// TIA Portal V19 export
FUNCTION "FC_EM_General" : Void   // FC1, FBD
TITLE = FC Algemeen
{ S7_Optimized_Access := 'TRUE' }
// stored: SetENOAutomatically false
   VAR_TEMP
      xFlashPeriod : Real;
   END_VAR
BEGIN

REGION Network 1: ------------------------------------------------------------------------ Inputs ------------------------------------------------------------------------
END_REGION

REGION Network 2: Verwerken van iStsNoodstop
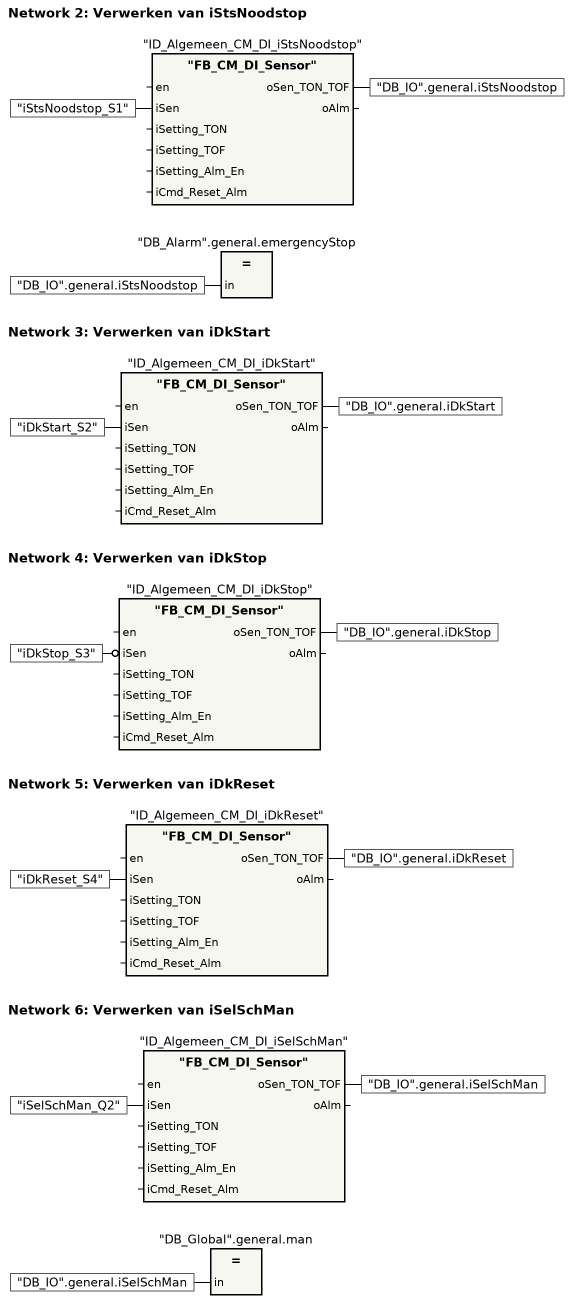
   "ID_Algemeen_CM_DI_iStsNoodstop"(iSen := "iStsNoodstop_S1", oSen_TON_TOF => "DB_IO".general.iStsNoodstop);   // "FB_CM_DI_Sensor"
   "DB_Alarm".general.emergencyStop := "DB_IO".general.iStsNoodstop;
END_REGION

REGION Network 3: Verwerken van iDkStart
   "ID_Algemeen_CM_DI_iDkStart"(iSen := "iDkStart_S2", oSen_TON_TOF => "DB_IO".general.iDkStart);   // "FB_CM_DI_Sensor"
END_REGION

REGION Network 4: Verwerken van iDkStop
   "ID_Algemeen_CM_DI_iDkStop"(iSen := NOT "iDkStop_S3", oSen_TON_TOF => "DB_IO".general.iDkStop);   // "FB_CM_DI_Sensor"
END_REGION

REGION Network 5: Verwerken van iDkReset
   "ID_Algemeen_CM_DI_iDkReset"(iSen := "iDkReset_S4", oSen_TON_TOF => "DB_IO".general.iDkReset);   // "FB_CM_DI_Sensor"
END_REGION

REGION Network 6: Verwerken van iSelSchMan
   "ID_Algemeen_CM_DI_iSelSchMan"(iSen := "iSelSchMan_Q2", oSen_TON_TOF => "DB_IO".general.iSelSchMan);   // "FB_CM_DI_Sensor"
   "DB_Global".general.man := "DB_IO".general.iSelSchMan;
END_REGION

REGION Network 7: ------------------------------------------------------------------------ Logic -------------------------------------------------------------------------
END_REGION

REGION Network 8: Start/stop logica van de installatie
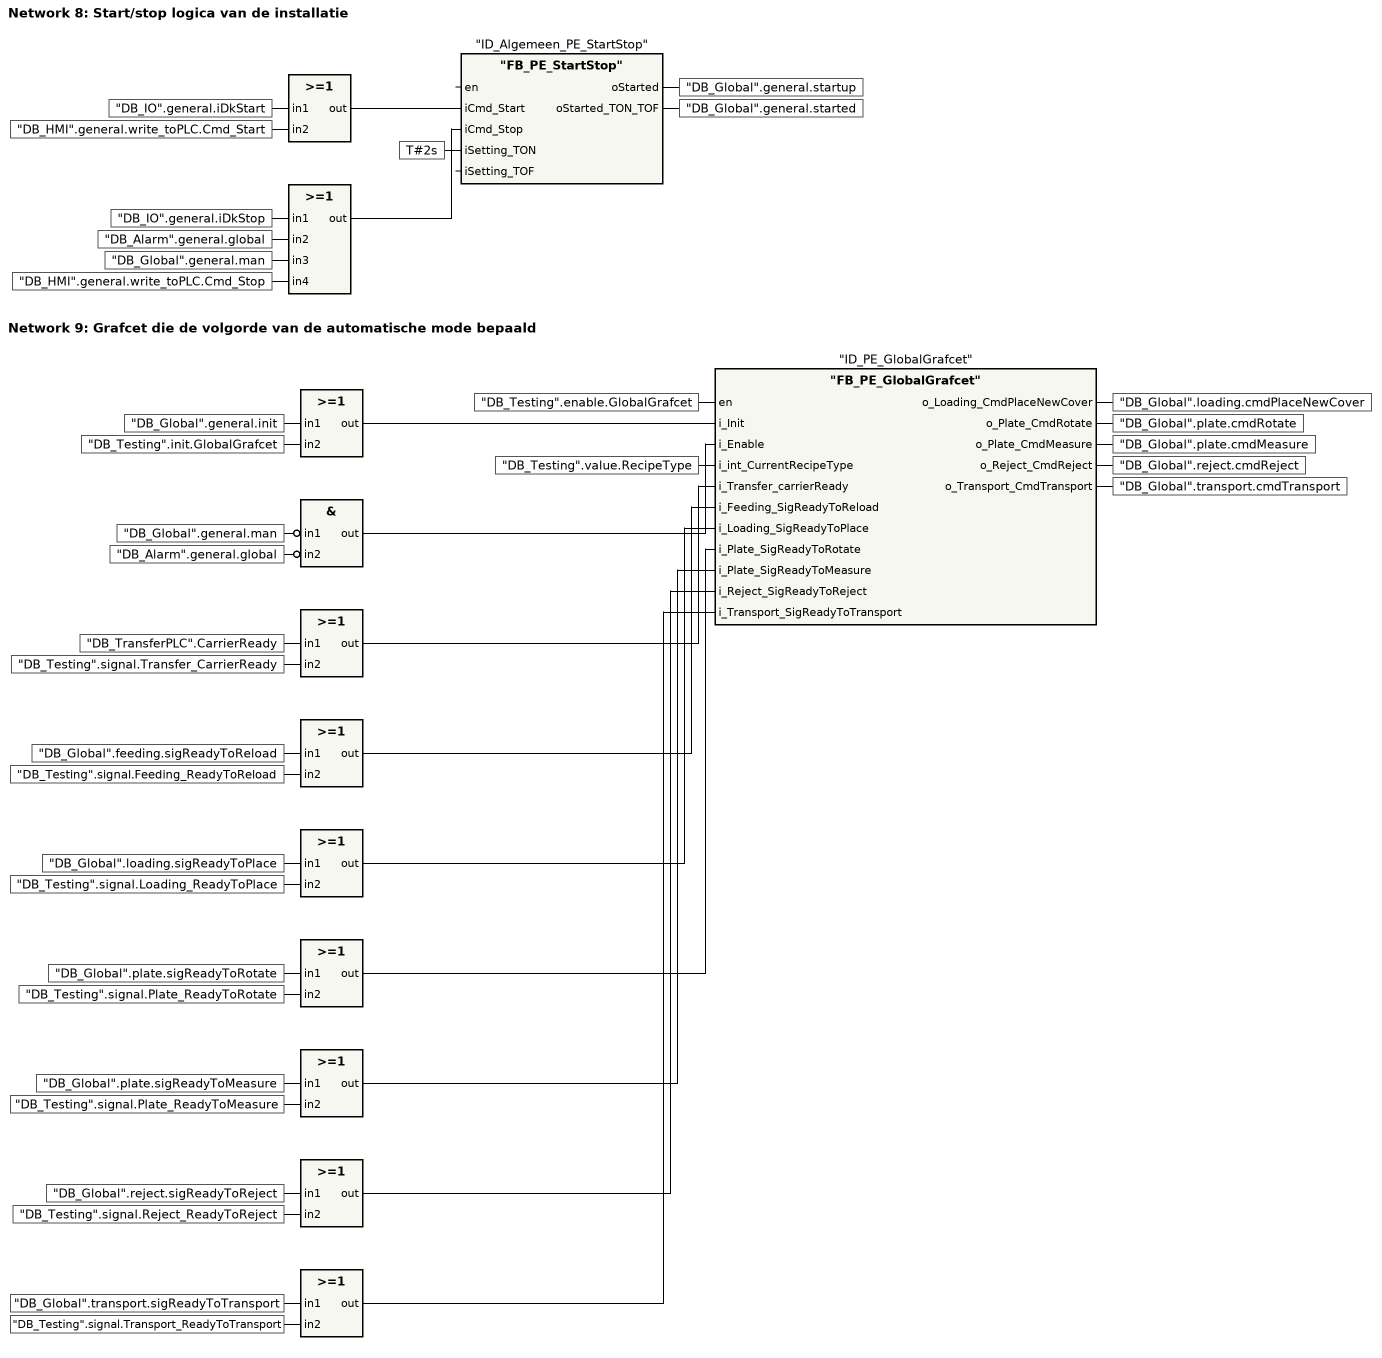
   "ID_Algemeen_PE_StartStop"(iCmd_Start := "DB_IO".general.iDkStart OR "DB_HMI".general.write_toPLC.Cmd_Start,   // "FB_PE_StartStop"
                           iCmd_Stop := "DB_IO".general.iDkStop OR "DB_Alarm".general.global OR "DB_Global".general.man OR "DB_HMI".general.write_toPLC.Cmd_Stop,
                           iSetting_TON := T#2s,
                           oStarted => "DB_Global".general.startup,
                           oStarted_TON_TOF => "DB_Global".general.started);
END_REGION

REGION Network 9: Grafcet die de volgorde van de automatische mode bepaald
   IF "DB_Testing".enable.GlobalGrafcet THEN
       "ID_PE_GlobalGrafcet"(i_Init := "DB_Global".general.init OR "DB_Testing".init.GlobalGrafcet,   // "FB_PE_GlobalGrafcet"
                             i_Enable := NOT "DB_Global".general.man AND NOT "DB_Alarm".general.global,
                             i_int_CurrentRecipeType := "DB_Testing".value.RecipeType,
                             i_Transfer_carrierReady := "DB_TransferPLC".CarrierReady OR "DB_Testing".signal.Transfer_CarrierReady,
                             i_Feeding_SigReadyToReload := "DB_Global".feeding.sigReadyToReload OR "DB_Testing".signal.Feeding_ReadyToReload,
                             i_Loading_SigReadyToPlace := "DB_Global".loading.sigReadyToPlace OR "DB_Testing".signal.Loading_ReadyToPlace,
                             i_Plate_SigReadyToRotate := "DB_Global".plate.sigReadyToRotate OR "DB_Testing".signal.Plate_ReadyToRotate,
                             i_Plate_SigReadyToMeasure := "DB_Global".plate.sigReadyToMeasure OR "DB_Testing".signal.Plate_ReadyToMeasure,
                             i_Reject_SigReadyToReject := "DB_Global".reject.sigReadyToReject OR "DB_Testing".signal.Reject_ReadyToReject,
                             i_Transport_SigReadyToTransport := "DB_Global".transport.sigReadyToTransport OR "DB_Testing".signal.Transport_ReadyToTransport,
                             o_Loading_CmdPlaceNewCover => "DB_Global".loading.cmdPlaceNewCover,
                             o_Plate_CmdRotate => "DB_Global".plate.cmdRotate,
                             o_Plate_CmdMeasure => "DB_Global".plate.cmdMeasure,
                             o_Reject_CmdReject => "DB_Global".reject.cmdReject,
                             o_Transport_CmdTransport => "DB_Global".transport.cmdTransport);
   END_IF;
END_REGION

REGION Network 10: ----------------------------------------------------------------------- Signals -----------------------------------------------------------------------
END_REGION

REGION Network 11: Genereren van reset puls
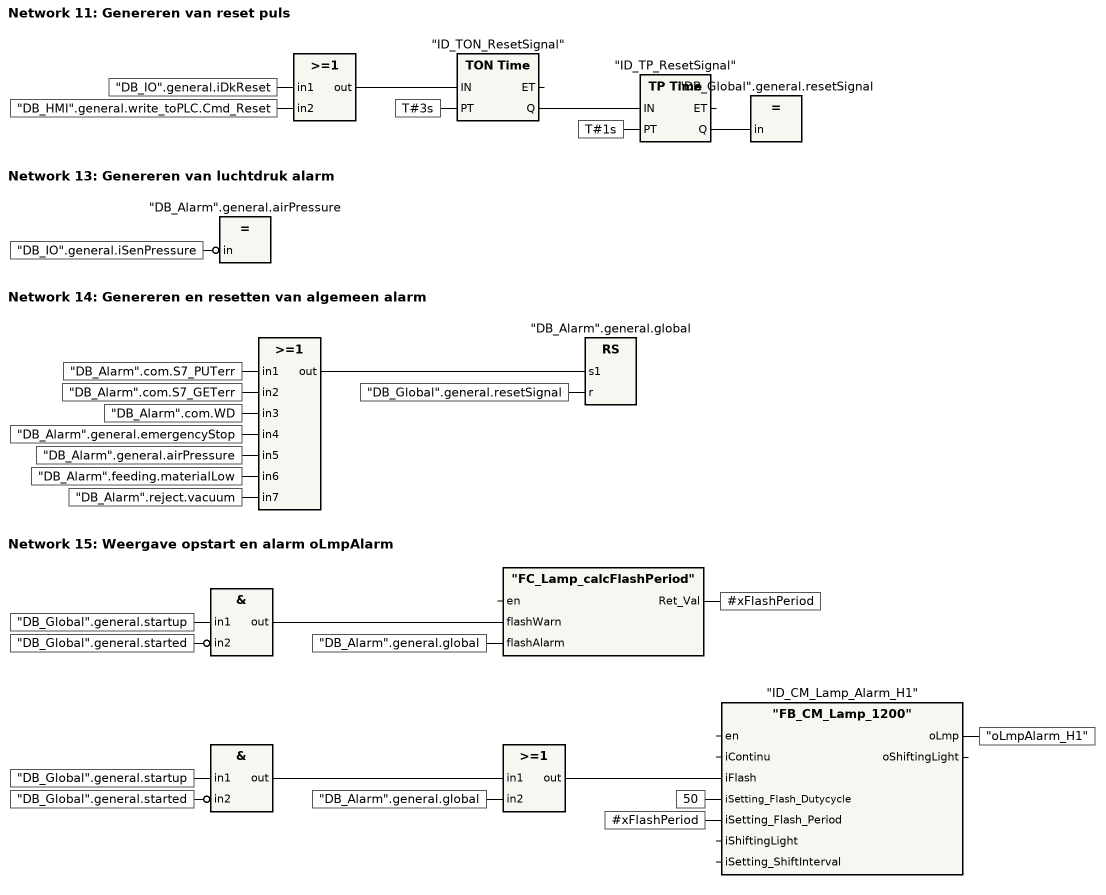
   "ID_TON_ResetSignal".TON(IN := "DB_IO".general.iDkReset OR "DB_HMI".general.write_toPLC.Cmd_Reset,
                           PT := T#3s);
   "ID_TP_ResetSignal".TP(IN := "ID_TON_ResetSignal".Q, PT := T#1s);
   "DB_Global".general.resetSignal := "ID_TP_ResetSignal".Q;
END_REGION

REGION Network 12: --------------------------------------------------------------------- Alarms ------------------------------------------------------------------------
END_REGION

REGION Network 13: Genereren van luchtdruk alarm
   "DB_Alarm".general.airPressure := NOT "DB_IO".general.iSenPressure;
END_REGION

REGION Network 14: Genereren en resetten van algemeen alarm
   IF "DB_Global".general.resetSignal THEN
       "DB_Alarm".general.global := FALSE;   // RS flip-flop
   END_IF;
   IF "DB_Alarm".com.S7_PUTerr OR "DB_Alarm".com.S7_GETerr OR "DB_Alarm".com.WD OR "DB_Alarm".general.emergencyStop OR "DB_Alarm".general.airPressure OR "DB_Alarm".feeding.materialLow OR "DB_Alarm".reject.vacuum THEN
       "DB_Alarm".general.global := TRUE;
   END_IF;
END_REGION

REGION Network 15: Weergave opstart en alarm oLmpAlarm
   #xFlashPeriod := "FC_Lamp_calcFlashPeriod"(flashWarn := "DB_Global".general.startup AND NOT "DB_Global".general.started,
                           flashAlarm := "DB_Alarm".general.global);
   "ID_CM_Lamp_Alarm_H1"(iFlash := ("DB_Global".general.startup AND NOT "DB_Global".general.started) OR "DB_Alarm".general.global,   // "FB_CM_Lamp_1200"
                         iSetting_Flash_Dutycycle := 50,
                         iSetting_Flash_Period := #xFlashPeriod,
                         oLmp => "oLmpAlarm_H1");
END_REGION
END_FUNCTION
